// TwinCAT 3 PLC project Start_Stop_Motor
// ProgramVersion: 3.1.4023.0
// libraries:
//   Tc2_MC2, * (Beckhoff Automation GmbH)
//   Tc2_MC2_Drive, * (Beckhoff Automation GmbH)
//   Tc2_Standard, * (Beckhoff Automation GmbH)
//   Tc2_System, * (Beckhoff Automation GmbH)
//   Tc3_Module, * (Beckhoff Automation GmbH)
// project tree:
//   DUTs/ ST_MC_Cmd.TcDUT, ST_MC_Status.TcDUT (not stored)
//   GVLs/ GVL_SA.TcGVL
//   / PlcTask.TcTTO
//   POUs/ MAIN.TcPOU, Motion.TcPOU
// real-time tasks:
//   TASK PlcTask: cycle T#10ms, priority 20, ADS port 350
// motion (NC):
//   TASK NC-Task 1 SAF: cycle T#2ms, priority 4, ADS port 501
//   TASK NC-Task 1 SVB: cycle T#10ms, priority 8, ADS port 511
//   AXIS Axis 1 (id 1)
//     OtherSettings: AllowMotionCmdToSlave=true
//     encoder EncType=1
//       Inc: RefSoftSyncMask=#x0000ffff
//     drive DrvType=24
//       Analog: TorqueSetpointScale=10, ScaleFactorActTorque=0.1
//       TimeComp: TaskDelayCycles=1
//     controller CtrType=1
//       CtrPara: PriorControlFactor=1
//         Observer: BandWidth=20
//   AXIS Virtual Axis (id 2)
//     OtherSettings: AllowMotionCmdToSlave=true
//     encoder EncType=1
//     drive DrvType=5
//       Analog: TorqueSetpointScale=10, ScaleFactorActTorque=0.1
//       TimeComp: TaskDelayCycles=1
//     controller CtrType=1
//       CtrPara: PriorControlFactor=1
//         Observer: BandWidth=20
// I/O:
//   DEVICE Device 1 (EtherCAT) (disabled), AmsNetId 5.71.198.244.2.1
//     Term 1 (EK1200) [EK1200-5000 EtherCAT Power supply (2A E-Bus)]
//       Term 2 (EL1008) [EL1008 8Ch. Dig. Input 24V, 3ms]
//       Term 3 (EL2008) [EL2008 8Ch. Dig. Output 24V, 0.5A]
//       Term 4 (EL3064) [EL3064 4Ch. Ana. Input 0-10V]
//       Term 5 (EL4002) [EL4002 2Ch. Ana. Output 0-10V, 12bit]
//       Term 6 (EL7031) [EL7031 1Ch. Stepper motor output stage (24V, 1.5A)]
//       Term 7 (EL9011) [EL9011 End Terminal]
// variable links:
//   NC-Task 1 SAF/Axes/Axis 1 <-> Device 1 (EtherCAT)/Term 1 (EK1200)/Term 6 (EL7031)
//     Drive/Inputs/In/nState1 @bit 3 <-> STM Status/Status/Error
//     Drive/Inputs/In/nState1 @bit 5 <-> STM Status/Status/Moving negative
//     Drive/Inputs/In/nState1 @bit 4 <-> STM Status/Status/Moving positive
//     Drive/Inputs/In/nState1 @bit 1 <-> STM Status/Status/Ready
//     Drive/Inputs/In/nState1 <-> STM Status/Status/Ready to enable
//     Drive/Inputs/In/nState1 @bit 6 <-> STM Status/Status/Torque reduced
//     Drive/Inputs/In/nState1 @bit 2 <-> STM Status/Status/Warning
//     Drive/Inputs/In/nState2 @bit 3 <-> STM Status/Status/Digital input 1
//     Drive/Inputs/In/nState2 @bit 4 <-> STM Status/Status/Digital input 2
//     Drive/Inputs/In/nState2 @bit 5 <-> STM Status/Status/Sync error
//     Drive/Inputs/In/nState2 @bit 7 <-> STM Status/Status/TxPDO Toggle
//     Drive/Inputs/In/nState4 @bit 1 <-> WcState/InputToggle
//     Drive/Inputs/In/nState4 <-> WcState/WcState
//     Drive/Outputs/Out/nCtrl1 <-> STM Control/Control/Enable
//     Drive/Outputs/Out/nCtrl1 @bit 2 <-> STM Control/Control/Reduce torque
//     Drive/Outputs/Out/nCtrl1 @bit 1 <-> STM Control/Control/Reset
//     Drive/Outputs/Out/nDataOut2[0] <-> STM Velocity/Velocity
//     Enc/Inputs/In/nDataIn1[0] <-> ENC Status compact/Counter value
//     Enc/Inputs/In/nDataIn2[0] <-> ENC Status compact/Latch value
//     Enc/Inputs/In/nState1 @bit 4 <-> ENC Status compact/Status/Counter overflow
//     Enc/Inputs/In/nState1 @bit 3 <-> ENC Status compact/Status/Counter underflow
//     Enc/Inputs/In/nState1 @bit 1 <-> ENC Status compact/Status/Latch extern valid
//     Enc/Inputs/In/nState1 @bit 2 <-> ENC Status compact/Status/Set counter done
//     Enc/Inputs/In/nState2 @bit 4 <-> ENC Status compact/Status/Status of extern latch
//     Enc/Inputs/In/nState2 @bit 5 <-> ENC Status compact/Status/Sync error
//     Enc/Inputs/In/nState2 @bit 7 <-> ENC Status compact/Status/TxPDO Toggle
//     Enc/Inputs/In/nState4 @bit 1 <-> WcState/InputToggle
//     Enc/Inputs/In/nState4 <-> WcState/WcState
//     Enc/Outputs/Out/nCtrl1 @bit 3 <-> ENC Control compact/Control/Enable latch extern on negative edge
//     Enc/Outputs/Out/nCtrl1 @bit 1 <-> ENC Control compact/Control/Enable latch extern on positive edge
//     Enc/Outputs/Out/nCtrl1 @bit 2 <-> ENC Control compact/Control/Set counter
//     Enc/Outputs/Out/nDataOut1[0] <-> ENC Control compact/Set counter value
//   Start Stop Motor/Start Stop Motor Instance <-> Device 1 (EtherCAT)/Term 1 (EK1200)/Term 2 (EL1008)
//     PlcTask Inputs/GVL_SA.bDigital_Inputs[1] <-> Channel 1/Input
//     PlcTask Inputs/GVL_SA.bDigital_Inputs[2] <-> Channel 2/Input
//   Start Stop Motor/Start Stop Motor Instance <-> Device 1 (EtherCAT)/Term 1 (EK1200)/Term 3 (EL2008)
//     PlcTask Outputs/GVL_SA.bDigital_Outputs[1] <-> Channel 1/Output
//     PlcTask Outputs/GVL_SA.bDigital_Outputs[2] <-> Channel 2/Output
//   Start Stop Motor/Start Stop Motor Instance <-> NC-Task 1 SAF/Axes/Virtual Axis
//     PlcTask Inputs/GVL_SA.singleAxis.NcToPlc <-> Outputs/ToPlc
//     PlcTask Outputs/GVL_SA.singleAxis.PlcToNc <-> Inputs/FromPlc

CONFIGURATION Start_Stop_Motor
    RESOURCE PLC ON TwinCAT3
        TASK PlcTask(INTERVAL := T#10ms, PRIORITY := 20);
        PROGRAM MAIN WITH PlcTask : MAIN;
    END_RESOURCE
END_CONFIGURATION

// ---- DUTs/ST_MC_Cmd.TcDUT
TYPE ST_MC_Cmd :
STRUCT
	bExe			: BOOL;
	lrVelocity		: LREAL;
	lrAcceleration	: LREAL;
	lrDeceleretion	: LREAL;
	lrJerk			: LREAL;
	lrDistance		: LREAL;
	lrPosition		: LREAL;
	EnuDirection	: MC_Direction;
	EnuBufferMode	: MC_BufferMode;
	EnuOptions		: ST_MoveOptions;
END_STRUCT
END_TYPE

// ---- GVLs/GVL_SA.TcGVL
{attribute 'qualified_only'}
VAR_GLOBAL
	bDigital_Inputs AT %I* : ARRAY[1..8] OF BOOL;
	bDigital_Outputs AT %Q* : ARRAY[1..8] OF BOOL;
	
	// Single Axis 'SA'
	singleAxis : AXIS_REF;
	
	// Motion Control Function Block instance variable 'fbSA'
	fbSA_Reset				: MC_RESET;
	fbSA_Power				: MC_POWER;
	fbSA_Home				: MC_HOME;
	fbSA_Jog				: MC_JOG;
	fbSA_Vel1				: MC_MoveVelocity;
	
	bSA_ResetExe			: BOOL;
	bSA_PowerEnCmd			: BOOL;
	bSA_PowerEnPositive		: BOOL;
	bSA_PowerEnNegative		: BOOL;
	
	bSA_HomeExe				: BOOL;
	bSA_HomeCamInput		: BOOL;
	
	bSA_JogFwd				: BOOL;
	bSA_JogRev				: BOOL;
	
	stSA_VelCmd1			: ST_MC_Cmd;
	stSA_VelCmd2			: ST_MC_Cmd;
	stSA_RelCmd1			: ST_MC_Cmd;
	stSA_RelCmd2			: ST_MC_Cmd;
	stSA_AbsCmd1			: ST_MC_Cmd;
	stSA_AbsCmd2			: ST_MC_Cmd;
	
	lrSA_PowerOverride		: LREAL;
	lrSA_HomePosition		: LREAL;
	lrSA_SetPosition		: LREAL;
	lrSA_JogVelocity		: LREAL;
	
	stSA_Reset				: ST_MC_Status;
	stSA_Power				: ST_MC_Status;
	stSA_Home				: ST_MC_Status;
	stSA_SetPosition		: ST_MC_Status;
	stSA_Jog				: ST_MC_Status;
	
	stSA_VelSts1			: ST_MC_Status;
	stSA_VelSts2			: ST_MC_Status;
	stSA_RelSts1			: ST_MC_Status;
	stSA_RelSts2			: ST_MC_Status;
	stSA_AbsSts1			: ST_MC_Status;
	stSA_AbsSts2			: ST_MC_Status;
	
END_VAR

// ---- POUs/MAIN.TcPOU
PROGRAM MAIN
VAR
END_VAR

Motion();

END_PROGRAM

// ---- POUs/Motion.TcPOU
PROGRAM Motion
VAR
END_VAR

Motion.StartStop();

METHOD SingleAxis_LD : BOOL
VAR_INPUT
END_VAR
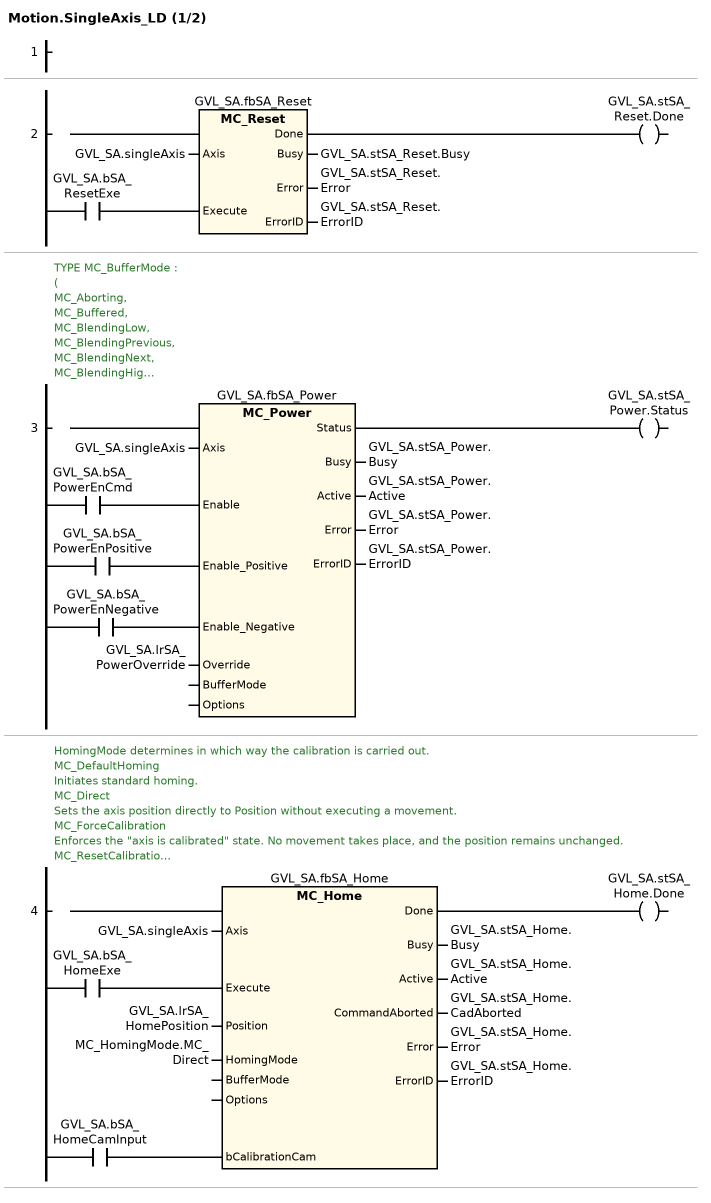
// NETWORK 1

// NETWORK 2
GVL_SA.fbSA_Reset(
    Axis := GVL_SA.singleAxis,
    Execute := GVL_SA.bSA_ResetExe,
    Busy => GVL_SA.stSA_Reset.Busy,
    Error => GVL_SA.stSA_Reset.Error,
    ErrorID => GVL_SA.stSA_Reset.ErrorID); // MC_Reset
GVL_SA.stSA_Reset.Done := GVL_SA.fbSA_Reset.Done;

// NETWORK 3
// TYPE MC_BufferMode :
// (
//     MC_Aborting,
//     MC_Buffered,
//     MC_BlendingLow,
//     MC_BlendingPrevious,
//     MC_BlendingNext,
//     MC_BlendingHigh
// );
// END_TYPE
GVL_SA.fbSA_Power(
    Axis := GVL_SA.singleAxis,
    Enable := GVL_SA.bSA_PowerEnCmd,
    Enable_Positive := GVL_SA.bSA_PowerEnPositive,
    Enable_Negative := GVL_SA.bSA_PowerEnNegative,
    Override := GVL_SA.lrSA_PowerOverride,
    Busy => GVL_SA.stSA_Power.Busy,
    Active => GVL_SA.stSA_Power.Active,
    Error => GVL_SA.stSA_Power.Error,
    ErrorID => GVL_SA.stSA_Power.ErrorID); // MC_Power
GVL_SA.stSA_Power.Status := GVL_SA.fbSA_Power.Status;

// NETWORK 4
// HomingMode determines in which way the calibration is carried out.
//
// MC_DefaultHoming
// Initiates standard homing.
// MC_Direct
// Sets the axis position directly to Position without executing a movement.
// MC_ForceCalibration
// Enforces the "axis is calibrated" state. No movement takes place, and the position remains unchanged.
// MC_ResetCalibration
// Resets the calibration state of the axis. No movement takes place, and the position remains unchanged.
GVL_SA.fbSA_Home(
    Axis := GVL_SA.singleAxis,
    Execute := GVL_SA.bSA_HomeExe,
    Position := GVL_SA.lrSA_HomePosition,
    HomingMode := MC_HomingMode.MC_Direct,
    bCalibrationCam := GVL_SA.bSA_HomeCamInput,
    Busy => GVL_SA.stSA_Home.Busy,
    Active => GVL_SA.stSA_Home.Active,
    CommandAborted => GVL_SA.stSA_Home.CadAborted,
    Error => GVL_SA.stSA_Home.Error,
    ErrorID => GVL_SA.stSA_Home.ErrorID); // MC_Home
GVL_SA.stSA_Home.Done := GVL_SA.fbSA_Home.Done;

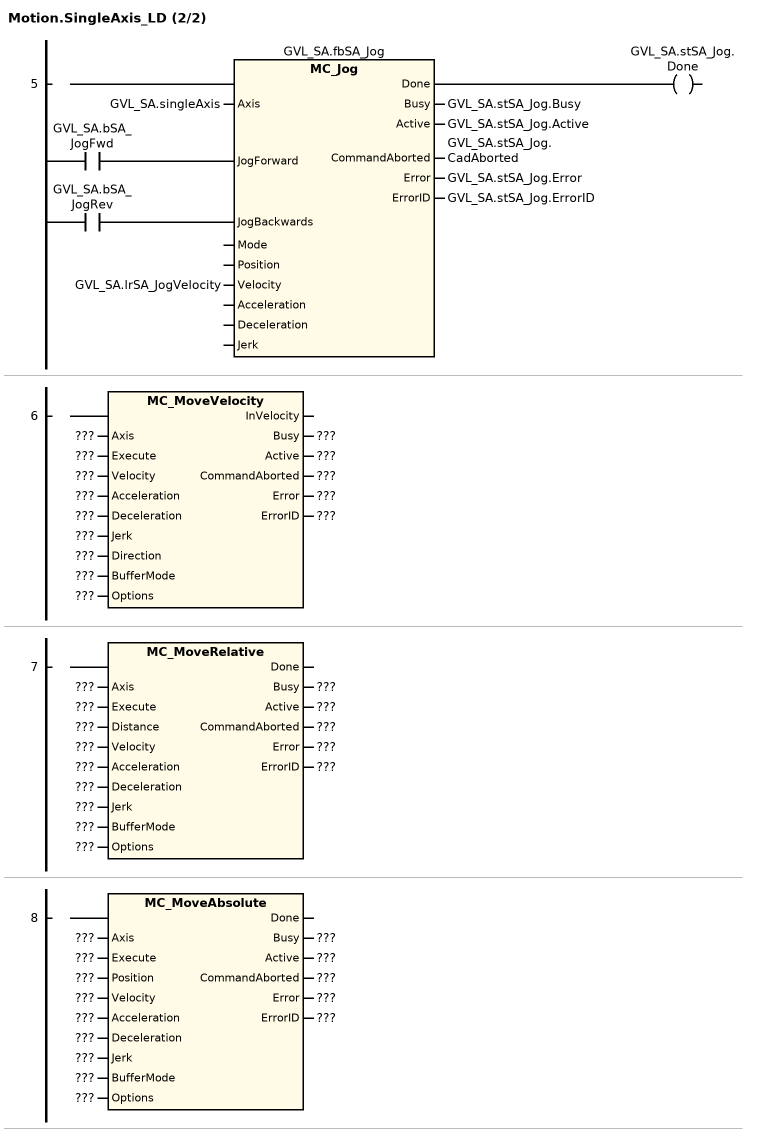
// NETWORK 5
GVL_SA.fbSA_Jog(
    Axis := GVL_SA.singleAxis,
    JogForward := GVL_SA.bSA_JogFwd,
    JogBackwards := GVL_SA.bSA_JogRev,
    Velocity := GVL_SA.lrSA_JogVelocity,
    Busy => GVL_SA.stSA_Jog.Busy,
    Active => GVL_SA.stSA_Jog.Active,
    CommandAborted => GVL_SA.stSA_Jog.CadAborted,
    Error => GVL_SA.stSA_Jog.Error,
    ErrorID => GVL_SA.stSA_Jog.ErrorID); // MC_Jog
GVL_SA.stSA_Jog.Done := GVL_SA.fbSA_Jog.Done;

// NETWORK 6
MC_MoveVelocity();

// NETWORK 7
MC_MoveRelative();

// NETWORK 8
MC_MoveAbsolute();
END_METHOD

METHOD StartStop : BOOL
VAR_INPUT
END_VAR
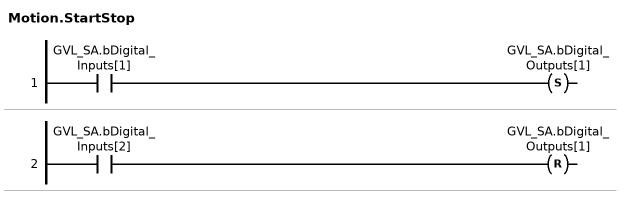
// NETWORK 1
GVL_SA.bDigital_Outputs[1] S= GVL_SA.bDigital_Inputs[1];

// NETWORK 2
GVL_SA.bDigital_Outputs[1] R= GVL_SA.bDigital_Inputs[2];
END_METHOD

END_PROGRAM
